INTERFACE ITF_PixelWritter

METHOD ClearPixelArrayCommand : BOOL
END_METHOD

METHOD CyclicLogic : BOOL
END_METHOD

METHOD ForwardCommandToFrameBuffer : BOOL
END_METHOD

METHOD ForwardExtCommandToFrame : BOOL
END_METHOD

METHOD SendCommandToPixelBuffer : BOOL
VAR_INPUT
	NewCommand: Command;
END_VAR
END_METHOD

METHOD SendExtCommand : BOOL
VAR_INPUT
	NewCommand: ExtendedCommand;
END_VAR
END_METHOD

END_INTERFACE

(* stored: Version 1.1.0.1, ProductVersion 3.1.4024.13
   Itf ITF_PixelWritter: Id {c677e114-1507-469b-8d59-eeb78b431049}
   Method ClearPixelArrayCommand: Id {dc4727ef-f7ca-4fb3-afe2-4d5de7a39dcd}
   Method CyclicLogic: Id {28a971d5-5c1f-42b4-a48c-b18be5431358}
   Method ForwardCommandToFrameBuffer: Id {30685db9-3a1b-440f-9b5e-1818fc352a0b}
   Method ForwardExtCommandToFrame: Id {54334c68-23d9-4ee6-8f2d-80748facd24b}
   Method SendCommandToPixelBuffer: Id {dfc29403-f450-410f-b163-d79ecec3e37f}
   Method SendExtCommand: Id {b1560dad-7075-4b7d-acb3-8b1876a355a4} *)
